# EPICS autosave request: tests/testfiles/cfg/SF_timing_us_PV.req
$(SYS).DESC
$(SYS)-Code-SP
$(SYS)-Delay-SP
$(SYS)-Freq-SP
